// LS Electric XG5000 project: 카운터
// PLC NewPLC
// module base 0 slot 0: 입출력 모듈:XBC-DR20S (DC 24V 입력 12점, 릴레이 출력 8점)

PROGRAM NewProgram (task: 스캔 프로그램)

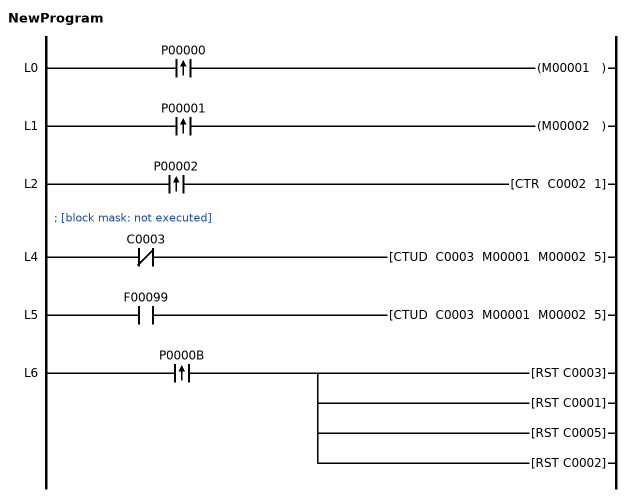
; L0
LOADP     P00000
OUT       M00001
; L1
LOADP     P00001
OUT       M00002
; L2
LOADP     P00002
CTR       C0002 1
; L4 (block mask: not executed)
LOAD NOT  C0003
CTUD      C0003 M00001 M00002 5
; L5
LOAD      F00099
CTUD      C0003 M00001 M00002 5
; L6
LOADP     P0000B
RST       C0003
RST       C0001
RST       C0005
RST       C0002